(* PLC project HW2TankController, iotrustlab-teaching HW2TankController 1.0 *)
(* stored: creationDateTime 2026-09-16T12:38:23, modificationDateTime 2026-09-16T12:38:23 *)

PROGRAM HW2TankController
  VAR_OUTPUT
    inlet_valve_open : BOOL := FALSE;
  END_VAR
  VAR
    reported_level_pct : REAL;
    LOW_LEVEL_PCT : REAL := 45.0;
    HIGH_LEVEL_PCT : REAL := 55.0;
  END_VAR

            IF reported_level_pct < LOW_LEVEL_PCT THEN
    inlet_valve_open := TRUE;
ELSIF reported_level_pct > HIGH_LEVEL_PCT THEN
    inlet_valve_open := FALSE;
END_IF;
          
END_PROGRAM

CONFIGURATION Config0
  RESOURCE Res0 ON PLC
    TASK task_HW2TankController(INTERVAL := T#100ms, PRIORITY := 0);
    PROGRAM HW2TankController_instance : HW2TankController;
  END_RESOURCE
END_CONFIGURATION
